(* PLC project fuse, Dassault Systèmes ControlBuild 2024x *)
(* stored: creationDateTime 2023-10-03T11:13:24-01:00 *)

(* This module simulates the trip of a fuse. This results in a power outage. *)
FUNCTION_BLOCK equipment_library.fuse
  VAR_INPUT
    energyBefore : BOOL := true;
    sensorSupply : BOOL := true;
  END_VAR
  VAR_OUTPUT
    fuseState : BOOL := false;
    energyAfter : BOOL := false;
  END_VAR
  VAR CONSTANT
    wiringLogic : BOOL := true;
  END_VAR
  VAR
    d_electric : BOOL := false;
    v_d_electric : BOOL := false;
  END_VAR


ACTION C_source_code:
/* ----------------------------------------------------------------	*/
/* Type : Model of Operative Behaviour					*/
/* Category :  Power								*/
/* Author : Dassault Systemes						*/
/* Update date : June 2018							*/
/* ----------------------------------------------------------------	*/
/* This module simulates the trip of a fuse.  				*/
/* This results in a power outage.						*/
/* It returns its state.							*/
/* ----------------------------------------------------------------	*/

/* ----------------------------------------------------------------	*/
/* Management of feedback to Control Part					*/
/*     if a fault is required, the fuse takes a preset state. 	*/
/*	if there is no power supply for sensors 				*/
/*         fuseState variable returns nothing				*/
/*     else fuseState variable returns fuse state combined with	*/
/*	    wiring logic (its default value is : positive).		*/
/* ----------------------------------------------------------------	*/
if (d_electric) fuseState = v_d_electric;
else
	if (sensorSupply) fuseState = sensorSupply ^ !wiringLogic;
	else fuseState = 0;

/* ----------------------------------------------------------------	*/
/* Management of the energy flow						*/
/*     Energy passes through the fuse if there is no electric fault.	*/
/* ----------------------------------------------------------------	*/
energyAfter = energyBefore & ! d_electric;
END_ACTION
END_FUNCTION_BLOCK
